// Mitsubishi GX Developer project: 16-301_20160505   PLC: FX1S

PROGRAM MAIN
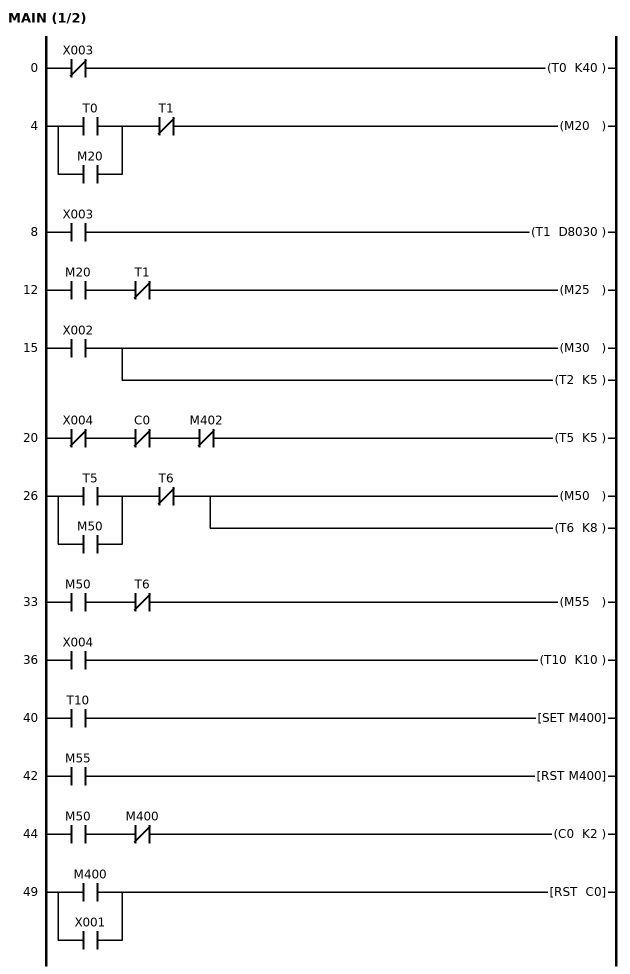
0     LDI     X003
      OUT     T0 K40
4     LD      T0
      OR      M20
      ANI     T1
      OUT     M20
8     LD      X003
      OUT     T1 D8030
12    LD      M20
      ANI     T1
      OUT     M25
15    LD      X002
      OUT     M30
      OUT     T2 K5
20    LDI     X004
      ANI     C0
      ANI     M402
      OUT     T5 K5
26    LD      T5
      OR      M50
      ANI     T6
      OUT     M50
      OUT     T6 K8
33    LD      M50
      ANI     T6
      OUT     M55
36    LD      X004
      OUT     T10 K10
40    LD      T10
      SET     M400
42    LD      M55
      RST     M400
44    LD      M50
      ANI     M400
      OUT     C0 K2
49    LD      M400
      OR      X001
      RST     C0
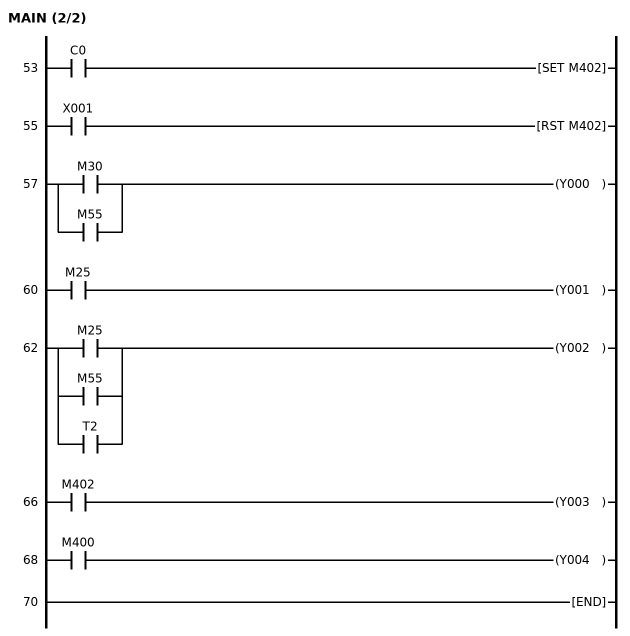
53    LD      C0
      SET     M402
55    LD      X001
      RST     M402
57    LD      M30
      OR      M55
      OUT     Y000
60    LD      M25
      OUT     Y001
62    LD      M25
      OR      M55
      OR      T2
      OUT     Y002
66    LD      M402
      OUT     Y003
68    LD      M400
      OUT     Y004
70    END
END_PROGRAM
